// TIA Portal V19 export
DATA_BLOCK "answer_from_drive_read"   // DB203
{ S7_Optimized_Access := 'TRUE' }
// stored: AutoNumber false, MemoryReserve 0
   VAR
      FaultBuffer : Array[1..16] of SinaParameter;
   END_VAR
BEGIN
END_DATA_BLOCK
